FUNCTION Sign : LREAL
VAR_INPUT
	Input:LREAL;
END_VAR
VAR
END_VAR

// sign符号函数
IF Input < 0 THEN
	Sign := -1;
ELSIF Input > 0 THEN
	Sign := 1;
ELSE Sign := 0;
END_IF

END_FUNCTION

(* stored: Version 1.1.0.1, ProductVersion 3.1.4024.11
   POU Sign: Id {cd5ce126-db14-471b-8312-e5d0b66d027f}, SpecialFunc None *)
